(* CoDeSys 2.3.9.50 project: Streaming.pro *)
(* Libraries: TcBase.lib 14.5.09 13:14:08, TcSystem.lib 7.6.16 12:01:22, TcEtherCAT.lib 30.11.16 20:52:18, STANDARD.LIB 5.6.98 13:03:02, TcUtilities.lib 3.2.16 17:08:58, C:\svn-sandbox\AR1500-Control\AR1500_Lib\AtlantisLib.lib 25.2.21 12:14:33 *)

(* Task configuration *)
TASK Standard (PRIORITY := 0, INTERVAL := T#10ms);
	MAIN
END_TASK

(* Global variable list: Global_Variables *)
VAR_GLOBAL CONSTANT
	MAX_BUFFER_SIZE: UDINT := 60000;
		gC_fPi : REAL := 3.141592654;
END_VAR
VAR_GLOBAL
END_VAR

(* Global variable list: TCS_Variables/C. Control/02_Pitch/Loads Test/GVL_LAT_Ctrl *)
VAR_GLOBAL
	visu_bNormalShutdown: BOOL;
	g_stHydairControl: Hydair_Data_Send;
	stVisuLoadSysCtrl: ST_LoadSysCtrl;
	stAutoLoadSysCtrl: ST_LoadSysCtrl;
	g_bConnectADSStream: BOOL:=TRUE;
	iCtrl: INT;
	sFilePath: STRING[75];
	sFilePathRcv: STRING[75];
	g_bVisuPauseFileStream: BOOL;
	g_bAutoPauseFileStream: BOOL;
	g_bAutoStartFileStream: BOOL;
	g_bVisuStartFileStream: BOOL;
	g_bVisuSelectFileStream: BOOL;
	g_bLoadProfileStreaming: BOOL;
	g_bDisableStreamToVPS:BOOL;   (*added to block stream data to VPS*)
	g_bDisableStreamToHCS:BOOL;   (*added to block stream data to HCS*)
	sTest_ID: STRING[15];
	g_bVisuLoadRampCmd: BOOL;
	g_bAutoLoadRampCmd: BOOL;
	g_bVisuStepLoadCmd: BOOL;
	g_bVisuStreamCmd:BOOL;
	arrTest: ARRAY [1..5] OF REAL;
	g_bVisuEnableVPSStream:BOOL;
	g_bVisuDisableVPSStream:BOOL;
	visu_bTestEFCTrip: BOOL;		(*buttpn to open the EFC safety relay by activating dq_B4_byPLC fed to the safety*)
END_VAR
VAR_GLOBAL RETAIN
	g_cMaxPositiveLoadLimit: REAL := 150;
	g_cMaxNegativeLoadLimit: REAL := -150;
	g_fLoadRampNegRateLimt: REAL;
	g_fLoadRampPosRateLimt: REAL;
END_VAR

(* Global variable list: TCS_Variables/C. Control/02_Pitch/Loads Test/GVL_LAT_Status *)
VAR_GLOBAL


	g_eFileStreamState:E_StreamState;

	g_fMZRam1LoadActualAv1s:REAL;	(*Load value Ram1 (MZ) after 1s average *)
	g_fMYRam2LoadActualAv1s:REAL;	(*Load value Ram1 (MY) after 1s average *)

	g_fRAM1LoadDemandFilteredADS:REAL;
	g_fRAM2LoadDemandFilteredADS:REAL;

         (*new vars*)
	g_nPitchTestMode:USINT;
	g_bPitchCtrlInterlock:BOOL;	(*interlock  for control of Pitch*)
	g_bLoadCtrlInterlock:BOOL; (*interlock signal for control of HCS*)
END_VAR
VAR_GLOBAL CONSTANT
	fCorrectionForRam1:REAL:=-0.2026;
	fCorrectionForRam2:REAL:=-1.8026;
	fCorrectionForRam3:REAL:=-4.0026;
END_VAR

(* Data type in C. Control/02_Pitch/Hydair Data *)
TYPE E_HydairState:
(
	eHCS_At_rest :=0,
	eHCS_CAN_Bus_Ready:=1,
	eHCS_Start_Hydraulics:=2,
	eHCS_Hydraulics_Ready:=3,
	eHCS_In_Operation:=4,
	eHCS_Passive:=5,
	eHCS_Manual_6,
	eHCS_Safety_Tripped:=7
);
END_TYPE

(* Data type in C. Control/02_Pitch/Hydair Data *)
TYPE E_MainState :
(
	STOP:=0,
	STARTING_HYDRAULICS:=1,
	HYDRAULICS_READY:=2,
	IN_OPERATION:=3,
	PASSIVE:=5,
	MANUAL:=6,
	SAFETY_TRIPPED:=7,
	SHUTDOWN:=8
);
END_TYPE

(* Data type in A. Operation_Ver2.10/01_Main_States *)
TYPE E_StateActivity :
(
	StEntry,
	StDo,
	StExit
);
END_TYPE

(* Data type in C. Control/02_Pitch/Test Rig *)
TYPE E_StreamState :
(
	e_streamState_Pause := 0,
	e_streamState_Start		:=1,
	e_streamState_Select	:=2
);
END_TYPE

(* Data type in C. Control/02_Pitch/Hydair Data *)
TYPE Hydair_Data_Rcv :
STRUCT
	stRam1_Sensors:Hydair_Ram_DataType;
	stRam2_Sensors:Hydair_Ram_DataType;
	stRam3_Sensors:Hydair_Ram_DataType;
	nFaultWord:UDINT;
	nInstrumentStatus:UINT;
	fHydr_Oil_Temp: REAL;
	bOilTempTooHigh:BOOL;
	bOfflineFilterClogged:BOOL;
	bHeartBeatEcho:BOOL;
	bMainPressureFilterClogged:BOOL;
	bMainReturnFilterClogged:BOOL;
	nHydairStateMachine:BYTE;
	bSafetyResetCmd:BOOL;
	bPassiveCtrlPermit:BOOL;
	bHydairReadyToOperate:BOOL;
	bHydairReadyToStartUp:BOOL;
	bEstopActive:BOOL;
	bActiveCtrlMode:BOOL;
END_STRUCT
END_TYPE

(* Data type in C. Control/02_Pitch/Hydair Data *)
TYPE Hydair_Data_Send :
STRUCT
	rRam1_LoadDemand:REAL;
	rRam2_LoadDemand:REAL;
	rRam3_LoadDemand:REAL;
	uiLoadsControl:ST_LoadSysCtrl;
END_STRUCT
END_TYPE

(* Data type in C. Control/02_Pitch/Hydair Data *)
TYPE Hydair_Ram_DataType :
STRUCT
	rLoad_Pin1: REAL;
	rAnnulusPressure:REAL;
	rFullBorePressure:REAL;
	rStroke:REAL;
	rLoadDemand:REAL;
	rLoadError:REAL;
END_STRUCT
END_TYPE

(* Data type in C. Control/02_Pitch/Hydair Data *)
TYPE J1939_Inputs :
STRUCT
	TxCounter  : UINT;
	RxCounter  : UINT;
	NoOfRxMessages   : UINT;
	RxMessage  : ARRAY [0..11] OF VARTYPE_EXTCANQUEUE;
(*	NodeState  : USINT;
	DiagFlag   : BOOL;*)
END_STRUCT
END_TYPE

(* Data type in C. Control/02_Pitch/Hydair Data *)
TYPE J1939_outputs :
STRUCT
	TxCounter : UINT;
	RxCounter   : UINT;
	NoOfTxMessages    : UINT;
	TxMessage  : ARRAY [0..1] OF VARTYPE_EXTCANQUEUE;
END_STRUCT
END_TYPE

(* Data type in C. Control/02_Pitch *)
TYPE PLCStruct :
STRUCT
	intVal : INT;
 	dintVal    : DINT;
	byteVal    : SINT;
	lrealVal  : LREAL;
	realVal  : REAL;
END_STRUCT
END_TYPE

(* Data type in C. Control/02_Pitch *)
TYPE ST_DataSetEntry :
STRUCT
	bFlag	: BOOL;
	nValue 	: REAL;
	sMsg 	: STRING(20) := 'Unknown';
END_STRUCT
END_TYPE

(* Data type in C. Control/02_Pitch/Hydair Data *)
TYPE ST_LoadSysCtrl :
STRUCT
	bDisablePassive: BOOL; (* Returns to AT_REST_POWER_ON *)
	rRam1_LoadDemand: REAL;
	rRam2_LoadDemand: REAL;
	rRam3_LoadDemand: REAL;
	bHeartbeat: BOOL;
	bStartUpCmd: BOOL; (* Start Hydraulics *)
	bOperateCmd: BOOL; (* Activate Load Control *)
	bPitchEFCActive: BOOL;
	bSafetyResetCmd: BOOL;
	bPassiveCtrlActive: BOOL;
	bGoToReady: BOOL;
	bGoToStop: BOOL;
	bRampDemand: BOOL;
	bStepDemand: BOOL;
	bStopCmd: BOOL; (* Stop Hydraulics *)
	bProfileStreamDemand: BOOL;
END_STRUCT
END_TYPE

(* Data type in C. Control/02_Pitch *)
TYPE stLoadData :
STRUCT
	sLoadID: STRING[30];
	rRig1_LoadDemand:REAL;
	rRig2_LoadDemand:REAL;
	rRig3_LoadDemand:REAL;
	rPitchAngleDemand:REAL;
	bStart:BOOL;
	bConnect:BOOL;
	bHeartbeat:BOOL;
END_STRUCT
END_TYPE

(* Data type in C. Control/02_Pitch/Hydair Data *)
TYPE VARTYPE_EXTCANQUEUE
STRUCT
	length: UINT;
	cobId: UDINT;
	rxData: ARRAY [0..7] OF USINT;
END_STRUCT
END_TYPE

(* POU MAIN, ST *)
PROGRAM MAIN
VAR
	fbReducePitchDutyCtrl:FB_ReducePitchDutyCtrl;

END_VAR
(*Manage profile streaming functions*)
P_LAT_Buffer_LoadData();
P_Manage_ADS_FileStream();

(*P_PitchReduceDutyCtrl();*)  (*Moved to function blocks*)
fbReducePitchDutyCtrl();
END_PROGRAM

(* POU Pitch Reduced Duty Cycle/FB_ReducePitchDutyCtrl, ST *)
FUNCTION_BLOCK FB_ReducePitchDutyCtrl
VAR_INPUT


	p_BetaDotSlow:REAL;                       (*Slow Pitch Rate Towards fine, imposed by Ramp function PItch_to_Fine state*)
	p_BetaNormal:REAL;

	p_tHysterysisBfeather:TIME; 	 (*Hysterysis time when moving towards feather*)


	p_tPitchAngleConstTime:TIME;	  (*time for Pitch rate to settle in Pitch_to_feather state before transition to Linger_1*)
	p_tLinger1Time:TIME;			  (*time for Linger1 state - increasing Pitch angle*)
	p_tLinger2Time:TIME;			  (*time for Linger2 state - decreasing Pitch*)

	bDisable:BOOL;   				(*always in NORMAL state when set*)
	rBetaDemandVSPR:REAL;           (*demand from VSPR*)
	rBetaActual:REAL;

	p_rPitchPosTol: REAL;			(*tolerance to the position reached flag use in Pitch_to_fine state*)
END_VAR


VAR_OUTPUT
	sState:STRING(20);
	rBetaMin:REAL;
END_VAR

VAR
	(*internals vars for state machine*)
	nState:USINT:=10;
	eStateActivity:E_StateActivity;
	nStep:USINT:=10;
	bFeathering:BOOL;
	tonPitchAngleConstTmr:TON;
	tonLinger1Timer:TON;
	tonLinger2Timer:TON;
	bPositionReached: BOOL;

	fbDeltaPitchFeather:FB_DeltaAlarm;
	fbDeltaPitchAngleConstant:FB_DeltaAlarm;
	tofBfeathering:TOF;
	rTrigRemove:R_TRIG;
	rTrigAdd:R_TRIG;
	rTrigGet:R_TRIG;
	rTrigReset:R_TRIG;

	fbRampBetaMin:FB_Ramp;



	(*VARS for Buffer Functions*)
        buffer  : ARRAY[0..1000] OF BYTE;
        fbStack : FB_MemStackBuffer;

        bReset  : BOOL := TRUE;
        bAdd    : BOOL := TRUE;
        bGet    : BOOL := TRUE;
        bRemove         : BOOL := TRUE;

        arrLast10BufferVals        : ARRAY[0..9] OF REAL;
        putEntry:REAL;
        getEntry        : REAL;
        i       : UDINT;
	instant: BOOL;


END_VAR
(*****************bFeathering***********************)
fbDeltaPitchFeather(
	tHysterysis:=T#2s ,		      (*ACTION: add input param*)
	rDeltaPosLim:=2 ,                           (*action: make ini-param*)
	rDeltaNegLim:=2 ,
	rValue:=rBetaActual ,
	bEnable:=1 ,
	bDeltaNegAlarm=> ,
	bDeltaPosAlarm=> ,
	rDelta=> );

tofBfeathering(IN:=fbDeltaPitchFeather.bDeltaPosAlarm , PT:=T#1s , Q=>bFeathering , ET=> );

(******************check Pitch angle constant in linger_2 state************************)

fbDeltaPitchAngleConstant(
	tHysterysis:=T#10ms ,
	rDeltaPosLim:=1 ,
	rDeltaNegLim:=1 ,
	rValue:= rBetaActual,
	bEnable:=(nState=30) ,
	bDeltaNegAlarm=> ,
	bDeltaPosAlarm=> ,
	rDelta=> );

tonPitchAngleConstTmr(IN:=(nSTate=20) AND NOT(fbDeltaPitchAngleConstant.bDeltaPosAlarm)   , PT:=p_tPitchAngleConstTime  );

A_BufferCommands();
A_StateMachine();
rTrigRemove(CLK:= , Q=>bRemove );
rTrigGet(CLK:= , Q=>bGet );
rTrigAdd(CLK:= , Q=> bAdd);
END_FUNCTION_BLOCK
ACTION A_BufferCommands:
IF bReset THEN(* Clear buffer *)
        bReset := FALSE;
        fbStack.A_Reset( pBuffer := ADR( buffer ), cbBuffer := SIZEOF( buffer ) );
END_IF

IF bAdd THEN(* Add entries *)
        bAdd := FALSE;

        fbStack.A_Push( pBuffer := ADR(buffer), cbBuffer := SIZEOF(buffer), pWrite := ADR(putEntry), cbWrite :=SIZEOF(putEntry) );
        IF fbStack.bOk THEN(* Success *)
                ;
        ELSE(* Buffer overflow *)
                ;
        END_IF

END_IF

IF bGet THEN(* Peek newest entry *)
        bGet := FALSE;
        fbStack.A_Top( pBuffer := ADR(buffer), cbBuffer := SIZEOF(buffer), pRead := ADR(getEntry), cbRead := SIZEOF(getEntry) );
        fbStack.A_Top( pBuffer := ADR(buffer), cbBuffer := SIZEOF(buffer), pRead := ADR(arrLast10BufferVals), cbRead := SIZEOF(arrLast10BufferVals) );
        IF fbStack.bOk THEN(* Success *)
                ;
        ELSE(* Buffer is empty *)
                ;
        END_IF
END_IF

IF bRemove THEN(* Remove newest entry *)
        bRemove := FALSE;
        fbStack.A_Pop( pBuffer := ADR(buffer), cbBuffer := SIZEOF(buffer), pRead := ADR(getEntry), cbRead := SIZEOF(getEntry) );
        IF fbStack.bOk THEN(* Success *)
                ;
        ELSE(* Buffer is empty *)
                ;
        END_IF
END_IF
END_ACTION
ACTION A_StateMachine:
CASE nState OF

	10:   (* NORMAL*)
		sState:='NORMAL';

		CASE eStateActivity OF
			StEntry:
				bReset:=1; (*reset buffer*)
				eStateActivity := StDo;
			StDo:
				rBetaMin:=p_BetaNormal;
				IF bFeathering THEN
					nState:=20;
					eStateActivity:=StEntry;
				END_IF
		END_CASE

	20:	(*PITCHING_TO_FEATHER*)
		sState:='PITCHING_TO_FEATHER';
		fbRampBetaMin.rNegRateLimit:=360;  (*limit movement to fine*)
		fbRampBetaMin.rPosRateLimit:=0; (*effectively no rate limit*)

		fbRampBetaMin.rStepCmd:=rBetaDemandVSPR;	(*set the step command to be VSPR Pitch demand*)

		rBetaMin:=fbRampBetaMin.rRampOutput;;


		IF bDisable THEN
			nState:=10;
		ELSIF tonPitchAngleConstTmr.Q THEN
			nState:=30;
		END_IF

	30:   (*LINGER_1*)
		sState:='LINGER_1';

		CASE eStateActivity OF
			StEntry:
				putEntry :=rBetaDemandVSPR;   (*assign the value sent to the buffer to be the Pitch Angle Demand from the VSPR*)
				rTrigAdd.CLK:=1; (*Add value to buffer*)
				rBetaMin:=rBetaDemandVSPR;
				eStateActivity := StDo;
			StDo:
				rTrigAdd.CLK:=0; (*Add value to buffer*)
				IF bDisable THEN
					nState:=10;
					eStateActivity:=StEntry;
				ELSIF tonLinger1Timer.Q THEN
					nState:=40;
					eStateActivity:=StEntry;
				ELSIF bFeathering THEN
					nState:=20;
					eStateActivity:=StEntry;
				END_IF
		END_CASE

	40:   (*PITCH_TO_FINE*)
		sState:='PITCH_TO_FINE';



		CASE nStep OF
			10:
				rTrigRemove.CLK:=1;    (*remove last record in buffer to make previous value current*)
				nStep:=20;

			20:
				rTrigRemove.CLK:=0;
				rTrigGet.CLK:=1;              (*get current value from buffer*)



				fbRampBetaMin.rStepCmd:=GetEntry;  (*assign current value of buffer to BetaMin*)

				nStep:=30;
			30:
				rTrigGet.CLK:=0;

				IF (rBetaActual >= (getEntry - p_rPitchPosTol)) AND (rBetaActual <= (getEntry + p_rPitchPosTol)) THEN
					bPositionReached:=1;
				ELSE
					bPositionReached:=0;
				END_IF

				IF bDisable OR NOT(fbStack.bOk) THEN   (*disable or Buffer empty*)
					nState:=10;
					nStep:=10;
				ELSIF bPositionReached THEN
					nState:=50;
					nStep:=10;
				ELSIF bFeathering THEN
					nState:=20;
					nStep:=10;
				END_IF

				IF fbStack.bOk THEN
					fbRampBetaMin.rPosRateLimit:=p_BetaDotSlow;
					fbRampBetaMin.rStepCmd:=getEntry;
					(*assign BetaMin the output of the ramp function*)
					rBetaMin:=fbRampBetaMin.rRampOutput;
				END_IF

		END_CASE

	50:  (*LINGER_2*)
		sState:='LINGER_2';


		IF bDisable THEN
			nState:=10;
		ELSIF tonLinger2Timer.Q THEN
			nState:=40;
		ELSIF bFeathering THEN
			nState:=20;
		END_IF

END_CASE;

tonLinger1Timer(IN:=(nState=30) , PT:=p_tLinger1Time);
tonLinger2Timer(IN:=(nState=50) , PT:=p_tLinger2Time );

fbRampBetaMin(
	rNegRateLimit:= ,
	rPosRateLimit:= ,
	rStepCmd:= ,
	rCurrentValue:=rBetaActual ,
	bRampActivated:=1 ,
	rRampOutput=> );
END_ACTION

(* POU Pitch Reduced Duty Cycle/FB_DeltaAlarm, ST *)
FUNCTION_BLOCK FB_DeltaAlarm
VAR_INPUT
	tHysterysis:TIME;
	rDeltaPosLim:REAL;
	rDeltaNegLim:REAL;
	rValue:REAL;
	bEnable:BOOL;
END_VAR

VAR_OUTPUT
	bDeltaNegAlarm:BOOL;
	bDeltaPosAlarm:BOOL;
	rDelta:REAL;
END_VAR

VAR
	nStep:USINT:=10;
	rValueSample:REAL;

	tonHysterysisTmr:TON;
END_VAR
(*if input for neg is pos, invert*)
IF rDeltaNegLim >0 THEN
	rDeltaNegLim:=rDeltaNegLim * (-1);
END_IF

(*calc delta between value sampled xn-1*)
rdelta := rValue-rValueSample;

(*start a timer when out of Hysterysis theshold*)
IF ((rDelta<=rDeltaNegLim) OR (rDelta>=rDeltaPosLim))  THEN
	tonHysterysisTmr.IN:=1;
	(*has signal been out threshold for tHysterysis time*)
	IF tonHysterysisTmr.Q THEN
		(*evaluate alarms*)
	 	bDeltaNegAlarm:= (rDelta<=rDeltaNegLim);
	 	bDeltaPosAlarm:= (rDelta>=rDeltaPosLim);
		rValueSample:=rValue;                                  (*Sample*);
	END_IF
ELSE
	(*reset Hysterysis timer if in Hysterysis theshold*)
	tonHysterysisTmr.IN:=0;
	bDeltaNegAlarm:= (rDelta<=rDeltaNegLim);
	 bDeltaPosAlarm:= (rDelta>=rDeltaPosLim);
END_IF

tonHysterysisTmr(PT:=tHysterysis );
END_FUNCTION_BLOCK

(* POU Pitch Reduced Duty Cycle/FB_Ramp, ST *)
FUNCTION_BLOCK FB_Ramp
VAR_INPUT
	rNegRateLimit:REAL;
	rPosRateLimit: REAL;
	rStepCmd: REAL;
	rCurrentValue:REAL;
	bRampActivated:BOOL;
END_VAR
VAR_OUTPUT
	rRampOutput: REAL;
END_VAR
VAR
	rRampIncrement: REAL;
	fbRampStartRTrig: R_TRIG;
END_VAR
(*COMPUTE RAMP SETPOINT*)

(*Initialise ramp to current position*)
fbRampStartRTrig(CLK:=bRampActivated);
IF fbRampStartRTrig.Q THEN rRampOutput := rCurrentValue; END_IF

(*Run ramp*)
IF bRampActivated THEN

	(*Compute cycle increment for ramp function*)
	IF rRampOutput < rStepCmd THEN
		rRampIncrement := F_rTaskCycleTime_s() * rNegRateLimit;
	ELSIF rRampOutput > rStepCmd THEN
		rRampIncrement := -1* F_rTaskCycleTime_s() * rPosRateLimit;
	END_IF

	(*If positiion error is within one ramp increment then set setpoint as final reference*)
	IF ABS(rStepCmd-rRampOutput) < ABS(rRampIncrement) THEN
		rRampOutput := rStepCmd;
	ELSE
		rRampOutput := rRampOutput + rRampIncrement;
	END_IF

(*If not ramp active then set demand to previous pitch angle cmd - hard stop*)
(*ELSIF NOT bSineActivated THEN
	rPositionSetpoint := rPositionSetpointPrev;*)
END_IF
END_FUNCTION_BLOCK

(* POU C. Control/02_Pitch_System/A. Operation/08_Speed_Sensing/F_rTaskCycleTime_s, ST *)
FUNCTION F_rTaskCycleTime_s : REAL
VAR
	rTime: REAL;
END_VAR
rTime := UDINT_TO_REAL(SystemTaskInfoArr[1].CycleTime);
F_rTaskCycleTime_s :=  rTime / 10000000.0;
END_FUNCTION

(* POU C. Control/Profile Streaming/P_LAT_Buffer_LoadData, ST *)
PROGRAM P_LAT_Buffer_LoadData
VAR
	fbFifo 		: FB_DataSetFifo := ( bOverwrite := TRUE );
	newEntry	: ARRAY [1..5] OF REAL;
	oldEntry		: ARRAY [1..5] OF REAL;
	bSuccess	: BOOL;
	nCount		: UDINT;
	nLoad		: UDINT;
	bReset 		: BOOL := TRUE;
	bAdd 		: BOOL;
	bGet		: BOOL;
	bRemove	: BOOL;
	bStreaming:BOOL;
	rLastValue:REAL;
	y: UINT;
	rTrigAdd: R_TRIG;
	r_trigGet: R_TRIG;
	rOldEntry:REAL;
	uiCount:UINT;
	rFreqOutDataHz:REAL;
	n:UINT;
	countInputs:UINT;
	arrReals: ARRAY [1..100] OF REAL;
	arrInputs: ARRAY [1..100] OF REAL;
	arrReals1: ARRAY [1..100] OF REAL;
	i: USINT;
	oldEntry_2: ARRAY [1..5] OF REAL;
	srNload:SR;
	n1: UINT;
	sPrevTime:REAL;
	rTime:REAL;
	rTrigSelectLoadProfile: R_TRIG;
	bExecEvery2Cycles:BOOL;
	uiCycleCount: USINT;
	tpAutoPause:TP;
	tpAutoStart:TP;
	SRControlPause:SR;
END_VAR
(*when a new profile is selected, reset the buffer*)
rTrigSelectLoadProfile(CLK:=(g_eFileStreamState=e_streamState_Select));
bReset:=rTrigSelectLoadProfile.Q;

IF bReset THEN
	oldEntry_2[3]:=0;
	oldEntry_2[4]:=0;
	oldEntry_2[5]:=0;
	oldEntry_2[2]:=87;(*g_fPitchAngleFilteredDeg;*)
	bReset := FALSE;
	(* reset fifo (clear all entries) *)
	fbFifo.A_Reset(	in := newEntry, bOk=>bSuccess, nCount=> nCount, nLoad => nLoad );
	y:=0;
END_IF
IF countInputs >=100 THEN
	countInputs:=1;
END_IF

IF n>=100 THEN
	n:=1;
END_IF
IF n1>=100 THEN
	n1:=1;
END_IF

rTrigAdd();

(*compute frequency*)
IF rOldEntry<>oldEntry_2[1] THEN
	IF uiCount<>0 THEN
		rFreqOutDataHz := 1 / (uiCount * 0.01);
	END_IF
	rOldEntry := oldEntry_2[1];
	uiCount:=1;
ELSE
	uiCount:=uiCount+1;
END_IF

IF arrTest[1]<>sPrevTime THEN
	sPrevTime:=arrTest[1];
	newEntry:=arrTest;
	 bAdd:=1;
END_IF

(*Clock out a signal every 5 time tasks cycles=20Hz as per input time series*)
IF srNload.Q1 AND (uiCycleCount>=5) THEN
	bRemove:=1;
	bStreaming:=FALSE;
	uiCycleCount:=0;
END_IF
uiCycleCount:=uiCycleCount+1;


IF bAdd AND NOT  SRControlPause.Q1 THEN
	bAdd := FALSE;
	fbFifo.A_Add(	in := newEntry, bOk=>bSuccess, nCount=> nCount, nLoad => nLoad );
	countInputs:=countInputs+1;
	arrInputs[countInputs]:=newEntry[1];
END_IF


srNload.SET1:=(nLoad>1);
srNload.RESET:=(nLoad<=0);
srNload();

(*control ADS stream based on load to prevent overflow*)
g_bAutoPauseFileStream := (nLoad>=90);
g_bAutoStartFileStream := (nLoad<10) AND srNload.Q1;
(*if operator pause then stop add or remove -- this will also pause the stream in P_Manage_ADS_Stream*)
SRControlPause(SET1:=g_bVisuPauseFileStream , RESET:= g_bVisuStartFileStream );

IF bRemove AND NOT SRControlPause.Q1 THEN
	bRemove:= FALSE;
	bStreaming:=TRUE;
	(* remove oldest entry *)
	fbFifo.A_Remove( out => oldEntry_2, bOk => bSuccess, nCount => nCount, nLoad => nLoad );
	arrReals1[n1]:=oldEntry_2[1];
	n1:=n1+1;
END_IF
END_PROGRAM

(* POU C. Control/Function Blocks/FB_DataSetFifo, ST *)
FUNCTION_BLOCK FB_DataSetFifo
VAR
	Name: BOOL;
	arrBuffer: ARRAY[0..MAX_BUFFER_SIZE] OF BYTE; (* Buffer memory used by FB_MemRingBuffer function block *)
	fbBuffer: FB_MemRingBuffer;
END_VAR
VAR_INPUT
	bOverwrite: BOOL;
	in: ARRAY [1..5] OF REAL;
END_VAR
VAR_OUTPUT
	bOk: BOOL;
	nCount: UDINT;
	nLoad: UDINT;
	out: ARRAY [1..5] OF REAL;
END_VAR
;
END_FUNCTION_BLOCK
ACTION A_Add:
fbBuffer.A_AddTail( pWrite:= ADR( in ),
					cbWrite:= SIZEOF( in ),
					pBuffer:= ADR( arrBuffer ),
					cbBuffer:= SIZEOF( arrBuffer ),
					bOk=> bOk,
					nCount => nCount );


IF NOT bOk THEN (* overflow ? *)
	IF bOverwrite THEN
		fbBuffer.A_RemoveHead(); (* remove one oldest entry *)

		fbBuffer.A_AddTail( bOk => bOk, nCount => nCount );
	END_IF
END_IF



nLoad := (fbBuffer.cbSize * 100) / MAX_BUFFER_SIZE;
END_ACTION
ACTION A_Get:
fbBuffer.A_GetHead( pRead:= ADR( out ),
					cbRead:= SIZEOF( out ),
					pBuffer:= ADR( arrBuffer ),
					cbBuffer:= SIZEOF( arrBuffer ),
					bOk=> bOk,
					nCount => nCount );

nLoad := (fbBuffer.cbSize * 100) / MAX_BUFFER_SIZE;
END_ACTION
ACTION A_Remove:
fbBuffer.A_RemoveHead( 	pRead:= ADR( out ),
						cbRead:= SIZEOF( out ),
						pBuffer:= ADR( arrBuffer ),
						cbBuffer:= SIZEOF( arrBuffer ),
						bOk=> bOk,
						nCount => nCount );

nLoad := (fbBuffer.cbSize * 100) / MAX_BUFFER_SIZE;
END_ACTION
ACTION A_Reset:
MEMSET( ADR( arrBuffer ), 0, SIZEOF( arrBuffer ) ); (* reset (optional) internal buffer *)

fbBuffer.A_Reset( 	bOk=> bOk,
					nCount => nCount );

nLoad := (fbBuffer.cbSize * 100) / MAX_BUFFER_SIZE;
END_ACTION

(* POU C. Control/Profile Streaming/P_Manage_ADS_FileStream, ST *)
PROGRAM P_Manage_ADS_FileStream
VAR
	RESelectFile:R_TRIG;
	REStartStream:R_TRIG;
	REPauseStream:R_TRIG;
	FELoadProfileSelect:R_TRIG;
	SRSelectFile: SR;
	SRStartStream: SR;
	SRPauseStream: SR;

END_VAR
(*Send commands to Python ADS streamer*)
RESelectFile(CLK:=g_bVisuSelectFileStream);
REStartStream(CLK:=g_bVisuStartFileStream OR g_bAutoStartFileStream);
REPauseStream(CLK:=g_bVisuPauseFileStream OR g_bAutoPauseFileStream);
FELoadProfileSelect(CLK:=g_bLoadProfileStreaming);

(*latch rising edge triggers*)
SRSelectFile(SET1:=RESelectFile.Q, RESET:=REStartStream.Q OR REPauseStream.Q);
SRStartStream(SET1:=REStartStream.Q, RESET:=REPauseStream.Q OR RESelectFile.Q);
SRPauseStream(SET1:=REPauseStream.Q OR FELoadProfileSelect.Q, RESET:=RESelectFile.Q OR REStartStream.Q);

(*Send command to interrupt select file from GUI*)
IF SRSelectFile.Q1 THEN
	iCtrl:=2;
END_IF
(*start streaming load profile values*)
IF SRStartStream.Q1 THEN
	iCtrl:=1;
END_IF
(*pause streaming of load profile values*)
IF SRPauseStream.Q1 THEN
	iCtrl:=0;
END_IF
(*map output state to enumeration*)
g_eFileStreamState:=iCtrl;
END_PROGRAM

(* POU Pitch Reduced Duty Cycle/P_PitchReducedDutyCtrl, ST *)
PROGRAM P_PitchReducedDutyCtrl
VAR
	fbReducePitchDutyCtrl:FB_ReducePitchDutyCtrl;
END_VAR
fbReducePitchDutyCtrl(
	p_BetaDotSlow:= 0.2,
	p_BetaNormal:= 1,
	p_tPitchAngleConstTime:=T#10s ,
	p_tLinger1Time:=T#10m ,
	p_tLinger2Time:= T#10m,
	bDisable:= ,
	rBetaDemandVSPR:= ,
	rBetaActual:= ,
	p_rPitchPosTol:= 0.2,
	sState=> ,
	rBetaMin=> );
END_PROGRAM

(* Visualisation VISU_CTRL_PROFILE
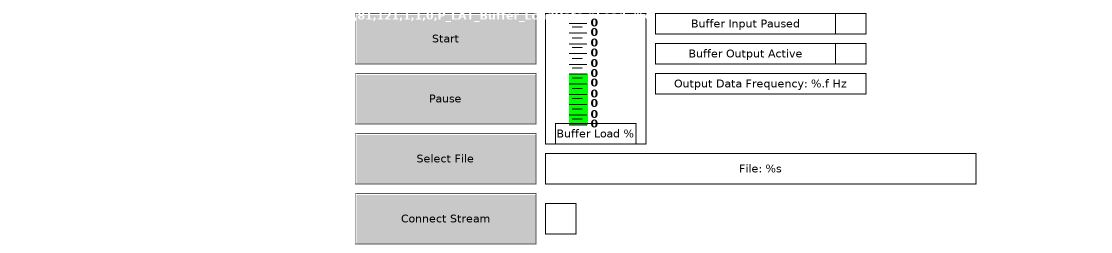
button at (10,20)-(191,71): text "Start"; taps g_bVisuStartFileStream
button at (10,80)-(191,131): text "Pause"; taps g_bVisuPauseFileStream
button at (10,140)-(191,191): text "Select File"; taps g_bVisuSelectFileStream
rectangle at (200,160)-(631,191): text "File: %s"; shows .sFilePath; editable
group at (210,20)-(291,141)
  rectangle at (0,2)-(1,3): text "{ExtendedElement},Visu\ElementDLL.ete,1,@Bargraph,81,121,1,1,0,P_LAT_Buffer_LoadData.nLoad,,%d,5,10,0,100,0,0,0,0,0,0,0,-13,16,700,Arial,0,255,0,255,0,0,0,0,0,0,0,0,0,,0,"
  rectangle at (13,62)-(30,114): alarm colour if (P_LAT_Buffer_LoadData.nLoad) < 0; top ((P_LAT_Buffer_LoadData.nLoad * 1.0) - 50)  * -1.04
  rectangle at (31,103)-(75,124): text "0"
  rectangle at (31,93)-(75,114): text "0"
  rectangle at (31,82)-(75,103): text "0"
  rectangle at (31,72)-(75,93): text "0"
  rectangle at (31,61)-(75,82): text "0"
  rectangle at (31,51)-(75,72): text "0"
  rectangle at (31,41)-(75,62): text "0"
  rectangle at (31,30)-(75,51): text "0"
  rectangle at (31,20)-(75,41): text "0"
  rectangle at (31,9)-(75,30): text "0"
  rectangle at (31,0)-(75,20): text "0"
rectangle at (310,20)-(491,41): text "Buffer Input Paused"
rectangle at (490,20)-(521,41): alarm colour if P_LAT_Buffer_LoadData.SRControlPause.Q1
rectangle at (310,50)-(491,71): text "Buffer Output Active"
rectangle at (490,50)-(521,71): alarm colour if P_LAT_Buffer_LoadData.srNload.SET1
rectangle at (310,80)-(521,101): text "Output Data Frequency: %.f Hz"; shows P_LAT_Buffer_LoadData.rFreqOutDataHz
rectangle at (210,130)-(291,151): text "Buffer Load %"
button at (10,200)-(191,251): text "Connect Stream"; toggles g_bConnectADSStream
rectangle at (200,210)-(231,241): alarm colour if g_bConnectADSStream
22 more shapes without text or variables
1 elements of other kinds (tables, trends, ...) not read
*)

(* Visualisation VISU_REDPITCHDUTY_CTRL
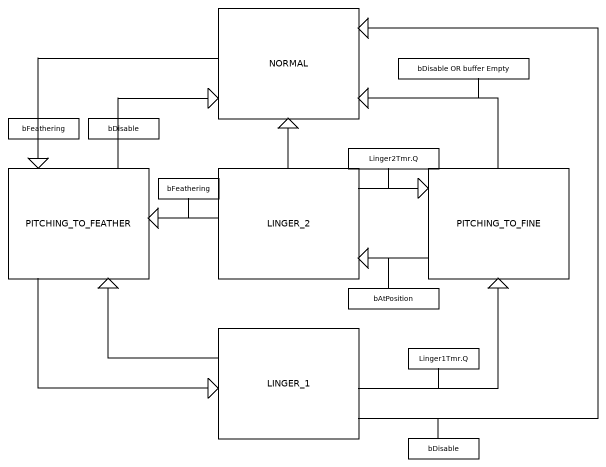
rectangle at (20,180)-(161,291): text "PITCHING_TO_FEATHER"
rectangle at (230,180)-(371,291): text "LINGER_2"
rectangle at (230,20)-(371,131): text "NORMAL"
rectangle at (440,180)-(581,291): text "PITCHING_TO_FINE"
rectangle at (230,340)-(371,451): text "LINGER_1"
rectangle at (420,450)-(491,471): text "bDisable"
rectangle at (420,360)-(491,381): text "Linger1Tmr.Q"
rectangle at (100,130)-(171,151): text "bDisable"
rectangle at (20,130)-(91,151): text "bFeathering"
rectangle at (360,160)-(451,181): text "Linger2Tmr.Q"
rectangle at (360,300)-(451,321): text "bAtPosition"
rectangle at (170,190)-(231,211): text "bFeathering"
rectangle at (410,70)-(541,91): text "bDisable OR buffer Empty"
27 more shapes without text or variables
1 elements of other kinds (tables, trends, ...) not read
*)
